(* PLC project Generated.project, CODESYS CODESYS V3.5 SP19 Patch 1 *)
(* stored: creationDateTime 2026-10-27T16:00:37.971314, modificationDateTime 2026-10-27T16:00:37.971314 *)

(* values of E_AutoCycleStep: AX0_REPOS: Repos / park : toutes commandes 0, etat neutre - etape initiale pure; AX1_INIT: Verif CONDITIONS INITIALES (Homed M1/M2, treuils FDC haut, M3 pas a droite de P1) - aucun mouvement, aucun referencement; AX2_TRANSLATE_P1: Translation vers P1 : joystick vers la droite, le cycle n'emet aucune commande M3 ; surveillance treuils au FDC haut; AX3_OPEN_BUCKET: Ouverture benne jusqu'au FDC logiciel benne ouverte --- DIVING (5 steps + retry) ---; AX4_DESCEND_DIVING: Plongee couplee benne ouverte palier 4 jusqu'a l'altimetrie de lancement (DiveStartMin_M) - Kobold PAS enclenche; AX5_KOBOLD_INIT: Activation contacteur Kobold << au vol >>, verif retour contacteur, descente palier 4 maintenue; AX6_SEARCH_IMMERSION: Recherche entree dans l'eau : attente front DI Kobold 0->1, descente palier 4 maintenue; AX7_SEARCH_BOTTOM: Recherche du fond : attente front DI Kobold 1->0, descente palier 4 maintenue; AX8_BOTTOM_CONFIRMED: Fond confirme : coupure instantanee treuils, set bit fond, TouchPositionM / RaiseTargetM --- EXTRACTION (4 steps) ---; AX9_RAISE_OFF_BOTTOM: Montee synchronisee : retendre les cables ; selecteur couplage BOTH/M1/M2 accessible; AX10_CLOSE_BUCKET: Fermeture benne, treuils explicitement 0; AX11_CTRL_ASCENT: Montee controle palier max reglable [1..2] + surveillance ecart vitesse M1/M2 ; benne mal fermee autorisee; AX12_LOADED_ASCENT: Montee en charge : palier 4 si benne fermee, palier 1 si mal fermee ; pas de ralenti 1 m avant top --- DECHARGE (6 steps) ---; AX13_DRAIN_PAUSE: Egouttage temporise - duree reglable IHM + bypass immediat; AX14_TRANSLATE_DUMP: Translation vers tremie (depart P1) + avertissements IHM; AX15A_DUMP_ARRIVE: Arrivee tremie : treuils a l'arret, attente geste operateur; AX15B_DUMP_OPEN: Vidage : ouverture benne au-dessus de la tremie, LES DEUX treuils a l'arret; AX15C_DUMP_REPOSITION: Repositionnement couple M1+M2 (option IHM maintenue), retour AX15B au relachement; AX18_DONE_SYNC: Fin de passe : compteur vidages + duree cycle ; msg << aller en P1 >> ; rebouclage direct sur AX2 --- STEPS SPECIAUX ---; AX_STAB: Repli defaut / stabilisation - pas une erreur; AX_DIVING_RETRY: Reprise diving : remontee assistee palier lent jusqu'au FDC haut puis retour AX4 ; sur erreur Kobold / joystick relache / palier <> 4 en AX5..AX7; AX3_WAIT_DIVE_START: Transition benne->plongee : sorties neutres jusqu'a l'arret mecanique confirme M1/M2, joystick pousse maintenu; AX10B_RACCORDEMENT_P1: Raccordement continu P1 fermeture benne -> montee controlee *)

{attribute 'qualified_only'}
{attribute 'strict'}
TYPE E_AutoCycleStep : (AX0_REPOS := 0, AX1_INIT := 1, AX2_TRANSLATE_P1 := 2, AX3_OPEN_BUCKET := 3, AX4_DESCEND_DIVING := 4, AX5_KOBOLD_INIT := 5, AX6_SEARCH_IMMERSION := 6, AX7_SEARCH_BOTTOM := 7, AX8_BOTTOM_CONFIRMED := 8, AX9_RAISE_OFF_BOTTOM := 9, AX10_CLOSE_BUCKET := 10, AX11_CTRL_ASCENT := 11, AX12_LOADED_ASCENT := 12, AX13_DRAIN_PAUSE := 13, AX14_TRANSLATE_DUMP := 14, AX15A_DUMP_ARRIVE := 15, AX15B_DUMP_OPEN := 16, AX15C_DUMP_REPOSITION := 17, AX18_DONE_SYNC := 18, AX_STAB := 19, AX_DIVING_RETRY := 20, AX3_WAIT_DIVE_START := 21, AX10B_RACCORDEMENT_P1 := 22);
END_TYPE
